/// Read integer values on RC
FUNCTION_BLOCK ReadIntegersFB EXTENDS RobotLibraryBaseFB
// ------------------------------------------------------------------------- 
//  SRCI Robot Library                                                
// ------------------------------------------------------------------------- 
//                                                                           
//  Object:      ReadIntegersFB                                       
//  Author:      Thorsten Brach                                                
//  Date:        2024-06-01
//
//  Description:                                              
//   
//                                                                           
//  Copyright: 
//    (C) 2024 Thorsten Brach. All rights reserved                                                                         
//                                                                           
//  Disclaimer:                                                                           
//    This project is provided without any guarantee and can be used for   
//    private and commercial purposes. Any commercial use is at the user’s 
//    own risk and responsibility.
//
// -------------------------------------------------------------------------
VAR_INPUT
  /// Start of the command at the rising edge
  Execute            : BOOL;
  /// Processing Mode
  ProcessingMode     : ProcessingMode;
  /// Specifies the desired target values that shall be read
  Index              : ARRAY[0..6] OF USINT; 
  /// Defines the target sequence in which the command will be executed
  SequenceFlag       : SequenceFlag;
  /// ID of associated trigger function:
  /// •  0: No Trigger (default)  No trigger related behavior
  /// • >0: Trigger - Start executing when the trigger function with the identical EmitterID is triggered.
  /// Always positive.
  /// For more information, see chapter 5.5.12 Triggers
  ListenerID         : SINT;
END_VAR
VAR_OUTPUT
  /// The command has been completed successfully
  Done               : BOOL;
  /// TRUE, while the following outputs return valid values:
  /// • Values
  Valid              : BOOL; 
  /// FB is being processed
  Busy               : BOOL;
  /// Command is transferred and confirmed by the RC
  CommandBuffered    : BOOL;
  /// The command was aborted by another command.
  CommandAborted     : BOOL;
  /// TRUE, while command is interrupted during execution and can be continued
  CommandInterrupted : BOOL;
  /// Receiving of input parameter values has been acknowledged by RC
  ParameterAccepted  : BOOL;
  /// Returned values of integer register
  Values             : ARRAY[0..6] OF INT;
  /// Unique system-generated ID of the "Action" when the function is triggered.
  /// • >0: The "Action" is started by the trigger function with identical FollowID.
  /// • <0: The "Action" is stopped by the trigger function with identical FollowID.
  /// For more information see chapter 5.5.12.4.
  OriginID           : USINT;
  /// Relates to ListenerID >0 
  /// Number of successful trigger -based command invocations
  /// For more information refer to chapter 5.5.12.4.
  InvocationCounter  : USINT;
END_VAR

                  
                

METHOD PROTECTED OnCall
VAR_IN_OUT
  /// Robot assignment of function
  AxesGroup         : AxesGroup; 
END_VAR
                        
                      
END_METHOD
END_FUNCTION_BLOCK

/// Read content of selected payload number
FUNCTION_BLOCK ReadLoadDataFB EXTENDS RobotLibraryBaseFB
// ------------------------------------------------------------------------- 
//  SRCI Robot Library                                                
// ------------------------------------------------------------------------- 
//                                                                           
//  Object:      ReadLoadDataFB                                       
//  Author:      Thorsten Brach                                                
//  Date:        2024-06-01
//
//  Description:                                              
//   
//                                                                           
//  Copyright: 
//    (C) 2024 Thorsten Brach. All rights reserved                                                                         
//                                                                           
//  Disclaimer:                                                                           
//    This project is provided without any guarantee and can be used for   
//    private and commercial purposes. Any commercial use is at the user’s 
//    own risk and responsibility.
//
// -------------------------------------------------------------------------
VAR_INPUT
  /// Start of the command at the rising edge
  Execute            : BOOL;
  /// Load index
  /// • -1: Currently used load on RC
  /// •  0: Not possible to read
  /// •  1 (default)..254: Load data
  LoadNo             : INT;
END_VAR
VAR_OUTPUT
  /// The command has been completed successfully
  Done               : BOOL;
  /// FB is being processed
  Busy               : BOOL;
  /// Command is transferred and confirmed by the RC
  CommandBuffered    : BOOL;
  /// Tool index
  LoadNoReturn       : USINT;
  /// Load data (see chapter 5.5.6.4)
  LoadData           : LoadData;
END_VAR

                  
                

METHOD PROTECTED OnCall
VAR_IN_OUT
  /// Robot assignment of function
  AxesGroup         : AxesGroup; 
END_VAR
                        
                      
END_METHOD
END_FUNCTION_BLOCK

/// Read error codes of pending errors and move them into user data block "RobotData"
FUNCTION_BLOCK ReadMessagesFB EXTENDS RobotLibraryBaseFB
// ------------------------------------------------------------------------- 
//  SRCI Robot Library                                                
// ------------------------------------------------------------------------- 
//                                                                           
//  Object:      ReadMessagesFB                                       
//  Author:      Thorsten Brach                                                
//  Date:        2024-06-01
//
//  Description:                                              
//   
//                                                                           
//  Copyright: 
//    (C) 2024 Thorsten Brach. All rights reserved                                                                         
//                                                                           
//  Disclaimer:                                                                           
//    This project is provided without any guarantee and can be used for   
//    private and commercial purposes. Any commercial use is at the user’s 
//    own risk and responsibility.
//
// -------------------------------------------------------------------------
VAR_INPUT
END_VAR
VAR_OUTPUT
END_VAR

                  
                

METHOD PROTECTED OnCall
VAR_IN_OUT
  /// Robot assignment of function
  AxesGroup         : AxesGroup; 
END_VAR
                        
                      
END_METHOD
END_FUNCTION_BLOCK

/// Read real values on RC
FUNCTION_BLOCK ReadRealsFB EXTENDS RobotLibraryBaseFB
// ------------------------------------------------------------------------- 
//  SRCI Robot Library                                                
// ------------------------------------------------------------------------- 
//                                                                           
//  Object:      ReadRealsFB                                       
//  Author:      Thorsten Brach                                                
//  Date:        2024-06-01
//
//  Description:                                              
//   
//                                                                           
//  Copyright: 
//    (C) 2024 Thorsten Brach. All rights reserved                                                                         
//                                                                           
//  Disclaimer:                                                                           
//    This project is provided without any guarantee and can be used for   
//    private and commercial purposes. Any commercial use is at the user’s 
//    own risk and responsibility.
//
// -------------------------------------------------------------------------
VAR_INPUT
  /// Start of the command at the rising edge
  Execute            : BOOL;
  /// Processing Mode
  ProcessingMode     : ProcessingMode;
  /// Specifies the desired target values that shall be read
  Index              : ARRAY[0..6] OF USINT; 
  /// Defines the target sequence in which the command will be executed
  SequenceFlag       : SequenceFlag;
  /// ID of associated trigger function:
  /// •  0: No Trigger (default)  No trigger related behavior
  /// • >0: Trigger - Start executing when the trigger function with the identical EmitterID is triggered.
  /// Always positive.
  /// For more information, see chapter 5.5.12 Triggers
  ListenerID         : SINT;
END_VAR
VAR_OUTPUT
  /// The command has been completed successfully
  Done               : BOOL;
  /// TRUE, while the following outputs return valid values:
  /// • Values
  Valid              : BOOL; 
  /// FB is being processed
  Busy               : BOOL;
  /// Command is transferred and confirmed by the RC
  CommandBuffered    : BOOL;
  /// The command was aborted by another command.
  CommandAborted     : BOOL;
  /// TRUE, while command is interrupted during execution and can be continued
  CommandInterrupted : BOOL;
  /// Receiving of input parameter values has been acknowledged by RC
  ParameterAccepted  : BOOL;
  /// Returned values of real register
  Values             : ARRAY[0..6] OF REAL;
  /// Unique system-generated ID of the "Action" when the function is triggered.
  /// • >0: The "Action" is started by the trigger function with identical FollowID.
  /// • <0: The "Action" is stopped by the trigger function with identical FollowID.
  /// For more information see chapter 5.5.12.4.
  OriginID           : USINT;
  /// Relates to ListenerID >0 
  /// Number of successful trigger -based command invocations
  /// For more information refer to chapter 5.5.12.4.
  InvocationCounter  : USINT;
END_VAR

                  
                

METHOD PROTECTED OnCall
VAR_IN_OUT
  /// Robot assignment of function
  AxesGroup         : AxesGroup; 
END_VAR
                        
                      
END_METHOD
END_FUNCTION_BLOCK

/// Read robot-specific data from the RC
FUNCTION_BLOCK ReadRobotDataFB EXTENDS RobotLibraryBaseFB
// ------------------------------------------------------------------------- 
//  SRCI Robot Library                                                
// ------------------------------------------------------------------------- 
//                                                                           
//  Object:      ReadRobotDataFB                                       
//  Author:      Thorsten Brach                                                
//  Date:        2024-06-01
//
//  Description:                                              
//   
//                                                                           
//  Copyright: 
//    (C) 2024 Thorsten Brach. All rights reserved                                                                         
//                                                                           
//  Disclaimer:                                                                           
//    This project is provided without any guarantee and can be used for   
//    private and commercial purposes. Any commercial use is at the user’s 
//    own risk and responsibility.
//
// -------------------------------------------------------------------------
VAR_INPUT
END_VAR
VAR_OUTPUT
END_VAR

                  
                

METHOD PROTECTED OnCall
VAR_IN_OUT
  /// Robot assignment of function
  AxesGroup         : AxesGroup; 
END_VAR
                        
                      
END_METHOD
END_FUNCTION_BLOCK

/// Read default values of dynamic parameters used by move commands
FUNCTION_BLOCK ReadRobotDefaultDynamicsFB EXTENDS RobotLibraryBaseFB
// ------------------------------------------------------------------------- 
//  SRCI Robot Library                                                
// ------------------------------------------------------------------------- 
//                                                                           
//  Object:      ReadRobotDefaultDynamicsFB                                       
//  Author:      Thorsten Brach                                                
//  Date:        2024-06-01
//
//  Description:                                              
//   
//                                                                           
//  Copyright: 
//    (C) 2024 Thorsten Brach. All rights reserved                                                                         
//                                                                           
//  Disclaimer:                                                                           
//    This project is provided without any guarantee and can be used for   
//    private and commercial purposes. Any commercial use is at the user’s 
//    own risk and responsibility.
//
// -------------------------------------------------------------------------
VAR_INPUT
  /// Start of the command at the rising edge
  Execute            : BOOL;
END_VAR

VAR_OUTPUT
  /// The command has been completed successfully
  Done               : BOOL;
  /// FB is being processed
  Busy               : BOOL;
  /// Command is transferred and confirmed by the RC
  CommandBuffered    : BOOL;
  /// Default dynamics values according to Table 6-148.
  DynamicValues      : DefaultDynamics;
END_VAR

                  
                

METHOD PROTECTED OnCall
VAR_IN_OUT
  /// Robot assignment of function
  AxesGroup         : AxesGroup; 
END_VAR
                        
                      
END_METHOD
END_FUNCTION_BLOCK

/// Read reference values of robot dynamics for path movement
FUNCTION_BLOCK ReadRobotReferenceDynamicsFB EXTENDS RobotLibraryBaseFB
// ------------------------------------------------------------------------- 
//  SRCI Robot Library                                                
// ------------------------------------------------------------------------- 
//                                                                           
//  Object:      ReadRobotReferenceDynamicsFB                                       
//  Author:      Thorsten Brach                                                
//  Date:        2024-06-01
//
//  Description:                                              
//   
//                                                                           
//  Copyright: 
//    (C) 2024 Thorsten Brach. All rights reserved                                                                         
//                                                                           
//  Disclaimer:                                                                           
//    This project is provided without any guarantee and can be used for   
//    private and commercial purposes. Any commercial use is at the user’s 
//    own risk and responsibility.
//
// -------------------------------------------------------------------------
VAR_INPUT
  /// Start of the command at the rising edge
  Execute            : BOOL;
END_VAR

VAR_OUTPUT
  /// The command has been completed successfully
  Done               : BOOL;
  /// FB is being processed
  Busy               : BOOL;
  /// Command is transferred and confirmed by the RC
  CommandBuffered    : BOOL;
  /// Reference dynamics values according to Table 6-109.
  DynamicValues      : ReferenceDynamics;
END_VAR

                  
                

METHOD PROTECTED OnCall
VAR_IN_OUT
  /// Robot assignment of function
  AxesGroup         : AxesGroup; 
END_VAR
                        
                      
END_METHOD
END_FUNCTION_BLOCK

/// Read actual software limits of the axes Positive and negative Limit of Joint J1…J6, E1…E6
FUNCTION_BLOCK ReadRobotSWLimitsFB EXTENDS RobotLibraryBaseFB
// ------------------------------------------------------------------------- 
//  SRCI Robot Library                                                
// ------------------------------------------------------------------------- 
//                                                                           
//  Object:      ReadRobotSWLimitsFB                                       
//  Author:      Thorsten Brach                                                
//  Date:        2024-06-01
//
//  Description:                                              
//   
//                                                                           
//  Copyright: 
//    (C) 2024 Thorsten Brach. All rights reserved                                                                         
//                                                                           
//  Disclaimer:                                                                           
//    This project is provided without any guarantee and can be used for   
//    private and commercial purposes. Any commercial use is at the user’s 
//    own risk and responsibility.
//
// -------------------------------------------------------------------------
VAR_INPUT
  /// Start of the command at the rising edge
  Execute            : BOOL;
END_VAR

VAR_OUTPUT
  /// The command has been completed successfully
  Done               : BOOL;
  /// FB is being processed
  Busy               : BOOL;
  /// Command is transferred and confirmed by the RC
  CommandBuffered    : BOOL;
  /// DLimits for joints and external axes according to Table 6-173.
  LimitValues        : SWLimits;
END_VAR

                  
                

METHOD PROTECTED OnCall
VAR_IN_OUT
  /// Robot assignment of function
  AxesGroup         : AxesGroup; 
END_VAR
                        
                      
END_METHOD
END_FUNCTION_BLOCK

/// Read specific parameter of the robot
FUNCTION_BLOCK ReadSystemVariableFB EXTENDS RobotLibraryBaseFB
// ------------------------------------------------------------------------- 
//  SRCI Robot Library                                                
// ------------------------------------------------------------------------- 
//                                                                           
//  Object:      ReadSystemVariableFB                                       
//  Author:      Thorsten Brach                                                
//  Date:        2024-06-01
//
//  Description:                                              
//   
//                                                                           
//  Copyright: 
//    (C) 2024 Thorsten Brach. All rights reserved                                                                         
//                                                                           
//  Disclaimer:                                                                           
//    This project is provided without any guarantee and can be used for   
//    private and commercial purposes. Any commercial use is at the user’s 
//    own risk and responsibility.
//
// -------------------------------------------------------------------------
VAR_INPUT
  /// Start of the command at the rising edge
  Execute            : BOOL;
  /// Processing Mode
  ProcessingMode     : ProcessingMode;
  /// Defines the parameter list which should be used:
  /// • FALSE: Standardized parameter list (default):
  ///          -  Read parameters on the RC based on a standardized parameter list
  /// • TRUE: Manufacturer specific parameter list:
  ///        -  Read parameters on the RC based on robot manufacturers-specific parameter lists
  RCParameter        : BOOL;
  /// Requested parameter ID in selected parameter list.
  /// •          0: undefined (default)
  /// • 1..65 535: Parameter ID
  ParameterID        : ARRAY[0..7] OF UINT;
  /// ID of the requested sub parameter in selected parameter list.
  /// • 0: ID 0 (default) (relates only to parameters without sub parameters)
  /// • 1..255: Indices 1 to 255 (relates only to parameters with sub parameters)
  SubParameterID     : ARRAY[0..7] OF USINT;
  /// Defines the target sequence in which the command will be executed
  SequenceFlag       : SequenceFlag;
  /// ID of associated trigger function:
  /// •  0: No Trigger (default)  No trigger related behavior
  /// • >0: Trigger - Start executing when the trigger function with the identical EmitterID is triggered.
  /// Always positive.
  /// For more information, see chapter 5.5.12 Triggers
  ListenerID         : SINT;
END_VAR
VAR_OUTPUT
  /// The command has been completed successfully
  Done               : BOOL;
  /// TRUE, while the following outputs return valid values:
  /// • DataType
  /// • Data_0
  /// • Data_1
  /// • Data_2
  /// • Data_3
  /// • Data_4
  /// • Data_5
  /// • Data_6
  /// • Data_7
  Valid              : BOOL; 
  /// FB is being processed
  Busy               : BOOL;
  /// Command is transferred and confirmed by the RC
  CommandBuffered    : BOOL;
  /// The command was aborted by another command.
  CommandAborted     : BOOL;
  /// TRUE, while command is interrupted during execution and can be continued
  CommandInterrupted : BOOL;
  /// Receiving of input parameter values has been acknowledged by RC
  ParameterAccepted  : BOOL;
  /// Parameter data type as specified in Table 6-613.
  DataType           : ARRAY[0..7] OF USINT;
  /// Parameter data addressed by input values of ParameterID[0] and SubParameterID[0]
  Data_0             : ARRAY[0..3] OF BYTE;
  /// Parameter data addressed by input values of ParameterID[1] and SubParameterID[1]
  Data_1             : ARRAY[0..3] OF BYTE;
  /// Parameter data addressed by input values of ParameterID[2] and SubParameterID[2]
  Data_2             : ARRAY[0..3] OF BYTE;
  /// Parameter data addressed by input values of ParameterID[3] and SubParameterID[3]
  Data_3             : ARRAY[0..3] OF BYTE;
  /// Parameter data addressed by input values of ParameterID[4] and SubParameterID[4]
  Data_4             : ARRAY[0..3] OF BYTE;
  /// Parameter data addressed by input values of ParameterID[5] and SubParameterID[5]
  Data_5             : ARRAY[0..3] OF BYTE;
  /// Parameter data addressed by input values of ParameterID[6] and SubParameterID[6]
  Data_6             : ARRAY[0..3] OF BYTE;
  /// Parameter data addressed by input values of ParameterID[7] and SubParameterID[7]
  Data_7             : ARRAY[0..3] OF BYTE;
  /// Unique system-generated ID of the "Action" when the function is triggered.
  /// • >0: The "Action" is started by the trigger function with identical FollowID.
  /// • <0: The "Action" is stopped by the trigger function with identical FollowID.
  /// For more information see chapter 5.5.12.4 EmitterID, ListenerID, FollowID and OriginID
  OriginID           : INT;
  /// Relates to ListenerID >0
  /// Number of successful trigger -based command invocations
  /// For more information refer to chapter 5.5.12.4.
  InvocationCounter  : USINT;
END_VAR

                  
                

METHOD PROTECTED OnCall
VAR_IN_OUT
  /// Robot assignment of function
  AxesGroup         : AxesGroup; 
END_VAR
                        
                      
END_METHOD
END_FUNCTION_BLOCK

/// Read content of selected tool number
FUNCTION_BLOCK ReadToolDataFB EXTENDS RobotLibraryBaseFB
// ------------------------------------------------------------------------- 
//  SRCI Robot Library                                                
// ------------------------------------------------------------------------- 
//                                                                           
//  Object:      ReadToolDataFB                                       
//  Author:      Thorsten Brach                                                
//  Date:        2024-06-01
//
//  Description:                                              
//   
//                                                                           
//  Copyright: 
//    (C) 2024 Thorsten Brach. All rights reserved                                                                         
//                                                                           
//  Disclaimer:                                                                           
//    This project is provided without any guarantee and can be used for   
//    private and commercial purposes. Any commercial use is at the user’s 
//    own risk and responsibility.
//
// -------------------------------------------------------------------------
VAR_INPUT
  /// Start of the command at the rising edge
  Execute            : BOOL;
  /// Tool index
  /// • -1: Currently used tool on RC
  /// •  0: Flange -  Not possible to change
  /// • 1 (default)..254: Tool Frame
  ToolNo             : INT;
END_VAR
VAR_OUTPUT
  /// The command has been completed successfully
  Done               : BOOL;
  /// FB is being processed
  Busy               : BOOL;
  /// Command is transferred and confirmed by the RC
  CommandBuffered    : BOOL;
  /// Tool index
  ToolNoReturn       : USINT;
  /// Tool data (see chapter 5.5.6.3)
  ToolData           : ToolData;
END_VAR

                  
                

METHOD PROTECTED OnCall
VAR_IN_OUT
  /// Robot assignment of function
  AxesGroup         : AxesGroup; 
END_VAR
                        
                      
END_METHOD
END_FUNCTION_BLOCK

/// Read configuration of defined work areas
FUNCTION_BLOCK ReadWorkAreaFB EXTENDS RobotLibraryBaseFB
// ------------------------------------------------------------------------- 
//  SRCI Robot Library                                                
// ------------------------------------------------------------------------- 
//                                                                           
//  Object:      ReadWorkAreaFB                                       
//  Author:      Thorsten Brach                                                
//  Date:        2024-06-01
//
//  Description:                                              
//   
//                                                                           
//  Copyright: 
//    (C) 2024 Thorsten Brach. All rights reserved                                                                         
//                                                                           
//  Disclaimer:                                                                           
//    This project is provided without any guarantee and can be used for   
//    private and commercial purposes. Any commercial use is at the user’s 
//    own risk and responsibility.
//
// -------------------------------------------------------------------------
VAR_INPUT
  /// Start of the command at the rising edge
  Execute                : BOOL;
  /// Index of the robot work area
  /// • 0 (default)..254
  WorkAreaNo             : USINT;
END_VAR
VAR_OUTPUT
  /// The command has been completed successfully
  Done                   : BOOL;
  /// FB is being processed
  Busy                   : BOOL;
  /// Command is transferred and confirmed by the RC
  CommandBuffered        : BOOL;
  /// Index of the robot work area
  WorkAreaNoReturn       : USINT;
  /// Data specific to the work area requested by Index.
  WorkAreaData           : RobotWorkArea;
END_VAR

                  
                

METHOD PROTECTED OnCall
VAR_IN_OUT
  /// Robot assignment of function
  AxesGroup         : AxesGroup; 
END_VAR
                        
                      
END_METHOD
END_FUNCTION_BLOCK

/// Move robot into contact with obstruction (mechanical Limit) and hold it in this position
FUNCTION_BLOCK SearchHardStopFB EXTENDS RobotLibraryBaseFB
// ------------------------------------------------------------------------- 
//  SRCI Robot Library                                                
// ------------------------------------------------------------------------- 
//                                                                           
//  Object:      SearchHardStopFB                                       
//  Author:      Thorsten Brach                                                
//  Date:        2024-06-01
//
//  Description:                                              
//   
//                                                                           
//  Copyright: 
//    (C) 2024 Thorsten Brach. All rights reserved                                                                         
//                                                                           
//  Disclaimer:                                                                           
//    This project is provided without any guarantee and can be used for   
//    private and commercial purposes. Any commercial use is at the user’s 
//    own risk and responsibility.
//
// -------------------------------------------------------------------------
VAR_INPUT
  /// Start of the command at the rising edge
  Execute            : BOOL;
  /// Absolute target coordinates in the selected coordinate system (see input parameters ToolNo and FrameNo)
  Position           : RobotCartesianPosition;
  /// Defines the type of collision detection, which parameter should be observed
  DetectionMode      : DetectionMode;
  /// Additional parameter for the detection of an end position. Defines the limits for seven joints, 
  /// where the robot stops when one of the limits is reached. Unit is depending on the "DetectionMode":
  /// • Torque (default) [Nm]  - Only positive values accepted
  /// • Force [N]              - Only positive values accepted
  /// • Electrical current [A] - Only positive values accepted
  /// • Following Error [mm]   - >0: Robot stops when the following error reached positive limit
  ///                          - <0: Robot stops when the following error reaches the negative limit
  DetectionVector    : ARRAY [0..6] OF REAL;
  /// TCP velocity in % of nominal velocity
  /// •  <0%: (default) - Use default velocity
  /// •   0%:           - Use internal minimal velocity
  /// • 100%:           - Use maximal reference velocity
  /// See chapter 5.5.7 Robot dynamics
  VelocityRate       : REAL;
  /// Acceleration for movement in % of nominal acceleration
  /// •  <0%: (default) - Use default acceleration
  /// •   0%:           - Use internal minimal acceleration
  /// • 100%:           - Use maximal reference acceleration
  /// See chapter 5.5.7 Robot dynamics
  AccelerationRate   : REAL;
  /// Deceleration for movement in % of nominal deceleration
  /// •  <0%: (default) - Use default deceleration 
  /// •   0%:           - Use internal minimal deceleration
  /// • 100%:           - Use maximal reference deceleration
  /// See chapter 5.5.7 Robot dynamics
  DecelerationRate   : REAL;
  /// Jerk of the movement in % of nominal jerk
  /// •  <0%: (default) - Use default jerk
  /// •   0%:           - Use internal minimal jerk
  /// • 100%:           - Use maximal reference jerk
  /// See chapter 5.5.7 Robot dynamics
  JerkRate           : REAL;
  /// Index of tool
  /// •      0: Flange (default)
  /// • 1..254: Tool frames
  ToolNo             : USINT;
  /// Index of frame
  /// •      0: WCS (default)
  /// • 1..254: User frames
  FrameNo            : USINT;
  /// Parameter which determines the behavior towards the previously sent and still active or buffered commands
  AbortingMode       : AbortingMode;
  /// Parameter to describe how the orientation axes (RX, RY, RZ) will be interpolated during the movement
  OriMode            : OriMode;
  /// Defines the usage of the config byte inside the position according to Table 6-238
  ConfigMode         : ArmConfigParameter;
  /// Defines the usage of the TurnNumber byte inside the position.
  TurnMode           : TurnMode;
  /// Set TRUE to allow manipulation of this move command through superimposing functions.
  /// For more information see chapter 5.5.9.5
  Manipulation       : BOOL;
  /// Defines the target sequence in which the command will be executed
  SequenceFlag       : SequenceFlag;
END_VAR

VAR_OUTPUT
  /// The command has been completed successfully
  Done               : BOOL;
  /// FB is being processed
  Busy               : BOOL;
  /// Command is transferred and confirmed by the RC
  CommandBuffered    : BOOL;
  /// The command takes control of the motion of the according axis group
  Active             : BOOL;
  /// The command was aborted by another command.
  CommandAborted     : BOOL;
  /// TRUE, while command is interrupted during execution and can be continued
  CommandInterrupted : BOOL;
  /// Distance-to-go of the current job.
  /// • -1: No valid value because move command is not yet active (valid values are pending) or not supported by RC
  /// • >0: Actual distance between current and target position
  /// •  0: Target position reached
  RemainingDistance  : REAL;
  /// Percentage of already traversed distance of current job.
  /// If not supported : • -1
  Progress           : REAL;
  /// The robot arm has detected an obstruction and stopped the movement
  InClamping         : BOOL;
END_VAR

                  
                

METHOD PROTECTED OnCall
VAR_IN_OUT
  /// Robot assignment of function
  AxesGroup         : AxesGroup; 
END_VAR
                        
                      
END_METHOD
END_FUNCTION_BLOCK

/// Move robot into contact with obstruction (mechanical Limit) and hold it in this position
FUNCTION_BLOCK SearchHardStopJFB EXTENDS RobotLibraryBaseFB
// ------------------------------------------------------------------------- 
//  SRCI Robot Library                                                
// ------------------------------------------------------------------------- 
//                                                                           
//  Object:      SearchHardStopJFB                                       
//  Author:      Thorsten Brach                                                
//  Date:        2024-06-01
//
//  Description:                                              
//   
//                                                                           
//  Copyright: 
//    (C) 2024 Thorsten Brach. All rights reserved                                                                         
//                                                                           
//  Disclaimer:                                                                           
//    This project is provided without any guarantee and can be used for   
//    private and commercial purposes. Any commercial use is at the user’s 
//    own risk and responsibility.
//
// -------------------------------------------------------------------------
VAR_INPUT
  /// Start of the command at the rising edge
  Execute            : BOOL;
  /// Absolute target coordinates in the selected coordinate system (see input parameters ToolNo and FrameNo)
  JointPosition      : RobotJointPosition;
  /// Defines the type of collision detection, which parameter should be observed
  DetectionMode      : DetectionMode;
  /// Additional parameter for the detection of an end position. Defines the limits for seven joints, 
  /// where the robot stops when one of the limits is reached. Unit is depending on the "DetectionMode":
  /// • Torque (default) [Nm]  - Only positive values accepted
  /// • Force [N]              - Only positive values accepted
  /// • Electrical current [A] - Only positive values accepted
  /// • Following Error [mm]   - >0: Robot stops when the following error reached positive limit
  ///                          - <0: Robot stops when the following error reaches the negative limit
  DetectionVector    : ARRAY [0..6] OF REAL;
  /// TCP velocity in % of nominal velocity
  /// •  <0%: (default) - Use default velocity
  /// •   0%:           - Use internal minimal velocity
  /// • 100%:           - Use maximal reference velocity
  /// See chapter 5.5.7 Robot dynamics
  VelocityRate       : REAL;
  /// Acceleration for movement in % of nominal acceleration
  /// •  <0%: (default) - Use default acceleration
  /// •   0%:           - Use internal minimal acceleration
  /// • 100%:           - Use maximal reference acceleration
  /// See chapter 5.5.7 Robot dynamics
  AccelerationRate   : REAL;
  /// Deceleration for movement in % of nominal deceleration
  /// •  <0%: (default) - Use default deceleration 
  /// •   0%:           - Use internal minimal deceleration
  /// • 100%:           - Use maximal reference deceleration
  /// See chapter 5.5.7 Robot dynamics
  DecelerationRate   : REAL;
  /// Jerk of the movement in % of nominal jerk
  /// •  <0%: (default) - Use default jerk
  /// •   0%:           - Use internal minimal jerk
  /// • 100%:           - Use maximal reference jerk
  /// See chapter 5.5.7 Robot dynamics
  JerkRate           : REAL;
  /// Index of tool
  /// •      0: Flange (default)
  /// • 1..254: Tool frames
  ToolNo             : USINT;
  /// Parameter which determines the behavior towards the previously sent and still active or buffered commands
  AbortingMode       : AbortingMode;
  /// Set TRUE to allow manipulation of this move command through superimposing functions.
  /// For more information see chapter 5.5.9.5
  Manipulation       : BOOL;
  /// Defines the target sequence in which the command will be executed
  SequenceFlag       : SequenceFlag;
END_VAR

VAR_OUTPUT
  /// The command has been completed successfully
  Done               : BOOL;
  /// FB is being processed
  Busy               : BOOL;
  /// Command is transferred and confirmed by the RC
  CommandBuffered    : BOOL;
  /// The command takes control of the motion of the according axis group
  Active             : BOOL;
  /// The command was aborted by another command.
  CommandAborted     : BOOL;
  /// TRUE, while command is interrupted during execution and can be continued
  CommandInterrupted : BOOL;
  /// Distance-to-go of the current job.
  /// • -1: No valid value because move command is not yet active (valid values are pending) or not supported by RC
  /// • >0: Actual distance between current and target position
  /// •  0: Target position reached
  RemainingDistance  : REAL;
  /// Percentage of already traversed distance of current job.
  /// If not supported : • -1
  Progress           : REAL;
  /// The robot arm has detected an obstruction and stopped the movement
  InClamping         : BOOL;
END_VAR

                  
                

METHOD PROTECTED OnCall
VAR_IN_OUT
  /// Robot assignment of function
  AxesGroup         : AxesGroup; 
END_VAR
                        
                      
END_METHOD
END_FUNCTION_BLOCK

/// Switch operation mode of RC (Automatic External, T1 External, T2 External)
FUNCTION_BLOCK SetOperationModeFB EXTENDS RobotLibraryBaseFB
// ------------------------------------------------------------------------- 
//  SRCI Robot Library                                                
// ------------------------------------------------------------------------- 
//                                                                           
//  Object:      SetOperationModeFB                                       
//  Author:      Thorsten Brach                                                
//  Date:        2024-06-01
//
//  Description:                                              
//   
//                                                                           
//  Copyright: 
//    (C) 2024 Thorsten Brach. All rights reserved                                                                         
//                                                                           
//  Disclaimer:                                                                           
//    This project is provided without any guarantee and can be used for   
//    private and commercial purposes. Any commercial use is at the user’s 
//    own risk and responsibility.
//
// -------------------------------------------------------------------------
VAR_INPUT
  /// Start of the command at the rising edge
  Execute                : BOOL;
  /// Limits for joints and external axes according to Table 6-180.
  OperationMode           : OperationMode;
END_VAR
VAR_OUTPUT
  /// The command has been completed successfully
  Done                   : BOOL;
  /// FB is being processed
  Busy                   : BOOL;
  /// Command is transferred and confirmed by the RC
  CommandBuffered        : BOOL;
END_VAR

                  
                

METHOD PROTECTED OnCall
VAR_IN_OUT
  /// Robot assignment of function
  AxesGroup         : AxesGroup; 
END_VAR
                        
                      
END_METHOD
END_FUNCTION_BLOCK

/// Set active sequence
FUNCTION_BLOCK SetSequenceFB EXTENDS RobotLibraryBaseFB
// ------------------------------------------------------------------------- 
//  SRCI Robot Library                                                
// ------------------------------------------------------------------------- 
//                                                                           
//  Object:      SetSequenceFB                                       
//  Author:      Thorsten Brach                                                
//  Date:        2024-06-01
//
//  Description:                                              
//   
//                                                                           
//  Copyright: 
//    (C) 2024 Thorsten Brach. All rights reserved                                                                         
//                                                                           
//  Disclaimer:                                                                           
//    This project is provided without any guarantee and can be used for   
//    private and commercial purposes. Any commercial use is at the user’s 
//    own risk and responsibility.
//
// -------------------------------------------------------------------------
VAR_INPUT
  /// Start of the command at the rising edge
  Execute         : BOOL;
  /// Defines sequence to be activated when function is executed
  TargetSequence  : SequenceFlag;
END_VAR

VAR_OUTPUT
  /// The command has been completed successfully
  Done            : BOOL;
  /// FB is being processed
  Busy            : BOOL;
  /// Command is transferred and confirmed by the RC
  CommandBuffered : BOOL;
END_VAR

                  
                

METHOD PROTECTED OnCall
VAR_IN_OUT
  /// Robot assignment of function
  AxesGroup         : AxesGroup; 
END_VAR
                        
                      
END_METHOD
END_FUNCTION_BLOCK

/// Create spline on RC from positions stored in PLC
FUNCTION_BLOCK CreateSplineFB EXTENDS RobotLibraryBaseFB
// ------------------------------------------------------------------------- 
//  SRCI Robot Library                                                
// ------------------------------------------------------------------------- 
//                                                                           
//  Object:      CreateSplineFB                                       
//  Author:      Thorsten Brach                                                
//  Date:        2024-06-01
//
//  Description:                                              
//   
//                                                                           
//  Copyright: 
//    (C) 2024 Thorsten Brach. All rights reserved                                                                         
//                                                                           
//  Disclaimer:                                                                           
//    This project is provided without any guarantee and can be used for   
//    private and commercial purposes. Any commercial use is at the user’s 
//    own risk and responsibility.
//
// -------------------------------------------------------------------------
VAR_INPUT
  /// Start of the command at the rising edge
  Execute         : BOOL;
  /// Define the method to calculate the path trajectory for the spline movement
  Mode            : SplineMode;
  /// Index of the spline trajectory to be created
  SplineID        : SINT;
  /// Contains all data relevant to the spline trajectory
  /// • Cartesian position
  /// • Coordinate systems
  /// • Dynamic parameters
  /// For more information refer to chapter 5.5.13.3
  SplineData      : ARRAY[1..RobotLibraryParameter.SPLINE_DATA_MAX] OF SplineData;
END_VAR
VAR_OUTPUT
  /// The command has been completed successfully
  Done            : BOOL;
  /// FB is being processed
  Busy            : BOOL;
  /// Command is transferred and confirmed by the RC
  CommandBuffered : BOOL;
END_VAR

                  
                

METHOD PROTECTED OnCall
VAR_IN_OUT
  /// Robot assignment of function
  AxesGroup         : AxesGroup; 
END_VAR
                        
                      
END_METHOD
END_FUNCTION_BLOCK

/// Delete spline previously created on RC
FUNCTION_BLOCK DeleteSplineFB EXTENDS RobotLibraryBaseFB
// ------------------------------------------------------------------------- 
//  SRCI Robot Library                                                
// ------------------------------------------------------------------------- 
//                                                                           
//  Object:      DeleteSplineFB                                       
//  Author:      Thorsten Brach                                                
//  Date:        2024-06-01
//
//  Description:                                              
//   
//                                                                           
//  Copyright: 
//    (C) 2024 Thorsten Brach. All rights reserved                                                                         
//                                                                           
//  Disclaimer:                                                                           
//    This project is provided without any guarantee and can be used for   
//    private and commercial purposes. Any commercial use is at the user’s 
//    own risk and responsibility.
//
// -------------------------------------------------------------------------
VAR_INPUT
  /// Start of the command at the rising edge
  Execute         : BOOL;
  /// Index of the spline trajectory to be deleted
  SplineID        : SINT;
END_VAR
VAR_OUTPUT
  /// The command has been completed successfully
  Done            : BOOL;
  /// FB is being processed
  Busy            : BOOL;
  /// Command is transferred and confirmed by the RC
  CommandBuffered : BOOL;
END_VAR

                  
                

METHOD PROTECTED OnCall
VAR_IN_OUT
  /// Robot assignment of function
  AxesGroup         : AxesGroup; 
END_VAR
                        
                      
END_METHOD
END_FUNCTION_BLOCK

/// Create and move spline on RC simultaneously
FUNCTION_BLOCK DynamicSplineFB EXTENDS RobotLibraryBaseFB
// ------------------------------------------------------------------------- 
//  SRCI Robot Library                                                
// ------------------------------------------------------------------------- 
//                                                                           
//  Object:      DynamicSplineFB                                       
//  Author:      Thorsten Brach                                                
//  Date:        2024-06-01
//
//  Description:                                              
//   
//                                                                           
//  Copyright: 
//    (C) 2024 Thorsten Brach. All rights reserved                                                                         
//                                                                           
//  Disclaimer:                                                                           
//    This project is provided without any guarantee and can be used for   
//    private and commercial purposes. Any commercial use is at the user’s 
//    own risk and responsibility.
//
// -------------------------------------------------------------------------
VAR_INPUT
  /// Start of the command at the rising edge
  Execute            : BOOL;
  /// Define the method to calculate the path trajectory for the spline movement
  Mode               : SplineMode;
  /// Parameter which determines the behavior towards the previously sent and still active or buffered commands
  AbortingMode       : AbortingMode;
  /// Parameter which determines the transition behavior at the end of the movement to be sent to the next command. 
  /// The user can choose a transition type between exact stop and different blend possibilities.
  BlendingMode       : BlendingMode;
  /// Additional parameter for the blending mode, to define i.e. velocity limit (%) or blending radius
  /// • [0]: default 10
  /// • [1]: default 0
  BlendingParameter  : ARRAY [0..1] OF REAL;
  /// Parameter is used if it is greater than 0 (default):
  /// • Velocity input is ignored
  /// • Parameter defines the time for the movement to reach the target position 
  /// Error is sent by the RC, if the time cannot be kept.
  MoveTime           : UINT;
  /// Contains all data relevant to the spline trajectory
  /// • Cartesian position
  /// • Coordinate systems
  /// • Dynamic parameters
  /// For more information refer to chapter 5.5.13.3
  SplineData         : ARRAY[1..RobotLibraryParameter.SPLINE_DATA_MAX] OF SplineData;
  /// Starts calculation and spline motion when equal or greater to number of buffered spline positions
  StartPosition      : INT; 
  /// Defines the target sequence in which the command will be executed
  SequenceFlag       : SequenceFlag;
END_VAR
VAR_OUTPUT
  /// FB is being processed
  Busy               : BOOL;
  /// Command is transferred and confirmed by the RC
  CommandBuffered    : BOOL;
  /// Function is enabled and new input values will be transmitted.
  Enabled            : BOOL;
  /// The command takes control of the motion of the according axis group
  Active             : BOOL;
  /// The command was aborted by another command.
  CommandAborted     : BOOL;
  /// TRUE, while command is interrupted during execution and can be continued.
  CommandInterrupted : BOOL;
  /// Receiving of input parameter values has been acknowledged by RC
  ParameterAccepted  : BOOL;
  /// Distance-to-go of the current job.
  /// • -1: No valid value because move command is not yet active (valid values are pending) or not supported by RC
  /// • >0: Actual distance between current and target position
  /// •  0: Target position reached 
  RemainingDistance  : REAL;
  /// Percentage of already traversed distance of actual segment of spline trajectory.
  /// If not supported: -1
  SegmentProgress    : REAL;
  /// Number of buffered, consecutive segments of spline trajectory. 
  Buffered           : INT;
  /// Number of calculated, consecutive segments of spline trajectory. Already calculated segments can no longer be modified.
  Calculated         : INT;
  /// Index of the currently active segment of spline data set.
  ActualIndex        : SINT;  
  /// Spline movement has been finished successfully. New SplineData will start a new spline movement.
  TrajectoryCompleted: BOOL;
END_VAR

                  
                

METHOD PROTECTED OnCall
VAR_IN_OUT
  /// Robot assignment of function
  AxesGroup         : AxesGroup; 
END_VAR
                        
                      
END_METHOD
END_FUNCTION_BLOCK

/// Call subprogram stored in RC from PLC
FUNCTION_BLOCK CallSubprogramFB EXTENDS RobotLibraryBaseFB
// ------------------------------------------------------------------------- 
//  SRCI Robot Library                                                
// ------------------------------------------------------------------------- 
//                                                                           
//  Object:      CallSubprogramFB                                       
//  Author:      Thorsten Brach                                                
//  Date:        2024-06-01
//
//  Description:                                              
//   
//                                                                           
//  Copyright: 
//    (C) 2024 Thorsten Brach. All rights reserved                                                                         
//                                                                           
//  Disclaimer:                                                                           
//    This project is provided without any guarantee and can be used for   
//    private and commercial purposes. Any commercial use is at the user’s 
//    own risk and responsibility.
//
// -------------------------------------------------------------------------
VAR_INPUT
  /// Start of the command at the rising edge
  Execute           : BOOL;
  /// Processing mode
  ProcessingMode    : ProcessingMode;
  /// Program number of the subprogram in the RC
  JobID             : UINT;
  /// Defines the target sequence in which the command will be executed
  SequenceFlag      : SequenceFlag;
  /// ID of associated trigger function:
  /// • 0: No Trigger (default) - No trigger related behavior
  /// • >0: Triggero - Start executing when the trigger function with the identical EmitterID is triggered.
  /// Always positive.
  /// For more information, see chapter 5.5.12 Triggers
  ListenerID        : SINT;
  /// Acyclic input parameters of the subprogram Array length adjusts to transmitted data (max 190 bytes)
  Data              : ARRAY[0..RobotLibraryParameter.SUB_PROGRAM_DATA_MAX] OF BYTE;
END_VAR

VAR_OUTPUT
  /// The command has been completed successfully
  Done               : BOOL;
  /// TRUE while the output ReturnData returns valid data according to the user defined subprogram
  Valid              : BOOL;
  /// FB is being processed
  Busy               : BOOL;
  /// Command is transferred and confirmed by the RC
  CommandBuffered    : BOOL;
  /// The requested subprogram on the RC is in progress. Movement of the axes trough this subprogram is possible.  
  InProgress         : BOOL;
  /// The command was aborted by another command
  CommandAborted     : BOOL;
  /// TRUE, while command is interrupted during execution and can be continued.
  CommandInterrupted : BOOL;
  /// Receiving of input parameter values has been acknowledged by RC
  ParameterAccepted  : BOOL;
  /// Unique, system-generated ID of the instance of CallSubprogram. 
  /// Can be used to specifically stop instance of a subprogram via the function Stop Subprogram (chapter 6.5.21) 
  /// if multiinstancing  is supported by RC 
  InstanceID         : DINT; 
  /// Percentage of already processed subprogram (must be configured by user)
  Progress           : REAL;
  /// Unique system-generated ID of the "Action" when the function is triggered.
  /// • >0: The "Action" is started by the trigger function with identical FollowID.
  /// • <0: The "Action" is stopped by the trigger function with identical FollowID.
  /// For more information see chapter 5.5.12.4 EmitterID, ListenerID, FollowID and OriginID
  OriginID           : INT;
  /// Relates to ListenerID >0
  /// Number of successful trigger -based command invocations
  /// For more information refer to chapter 5.5.12.4.
  InvocationCounter  : USINT;
  /// Acyclic output parameters of the subprogram Array length adjusts to transmitted data (max 190 bytes)
  ReturnData         : ARRAY[0..RobotLibraryParameter.SUB_PROGRAM_DATA_MAX] OF BYTE;
END_VAR

                  
                

METHOD PROTECTED OnCall
VAR_IN_OUT
  /// Robot assignment of function
  AxesGroup         : AxesGroup; 
END_VAR
                        
                      
END_METHOD
END_FUNCTION_BLOCK

/// Reads cyclic data of called subprogram
FUNCTION_BLOCK ReadCallSubprogramCyclicFB EXTENDS RobotLibraryBaseFB
// ------------------------------------------------------------------------- 
//  SRCI Robot Library                                                
// ------------------------------------------------------------------------- 
//                                                                           
//  Object:      ReadCallSubprogramCyclicFB                                       
//  Author:      Thorsten Brach                                                
//  Date:        2024-06-01
//
//  Description:                                              
//   
//                                                                           
//  Copyright: 
//    (C) 2024 Thorsten Brach. All rights reserved                                                                         
//                                                                           
//  Disclaimer:                                                                           
//    This project is provided without any guarantee and can be used for   
//    private and commercial purposes. Any commercial use is at the user’s 
//    own risk and responsibility.
//
// -------------------------------------------------------------------------
VAR_INPUT
  /// Set TRUE (default) to cyclically transmit data to the RC
  Enable            : BOOL;
END_VAR

VAR_OUTPUT
  /// Function is returning cyclic data from the RC
  Enabled           : BOOL;
  /// FB is being processed
  Busy              : BOOL;
  /// Cyclic input data of subprogram
  Data              : ARRAY[0..25] OF BYTE;
  
END_VAR

                  
                

METHOD PROTECTED OnCall
VAR_IN_OUT
  /// Robot assignment of function
  AxesGroup         : AxesGroup; 
END_VAR
                        
                      
END_METHOD
END_FUNCTION_BLOCK

/// Stops an active subprogram
FUNCTION_BLOCK StopSubprogramFB EXTENDS RobotLibraryBaseFB
// ------------------------------------------------------------------------- 
//  SRCI Robot Library                                                
// ------------------------------------------------------------------------- 
//                                                                           
//  Object:      StopSubprogramFB                                       
//  Author:      Thorsten Brach                                                
//  Date:        2024-06-01
//
//  Description:                                              
//   
//                                                                           
//  Copyright: 
//    (C) 2024 Thorsten Brach. All rights reserved                                                                         
//                                                                           
//  Disclaimer:                                                                           
//    This project is provided without any guarantee and can be used for   
//    private and commercial purposes. Any commercial use is at the user’s 
//    own risk and responsibility.
//
// -------------------------------------------------------------------------
VAR_INPUT
  /// Start of the command at the rising edge
  Execute           : BOOL;
  /// Processing mode
  ProcessingMode    : ProcessingMode;
  /// Defines how target subprogram is defined
  StopMode          : StopMode;
  /// JobID or InstanceID of target subprogram according to selected StopMode
  /// • Refers to StopMode 0 (Stop via JobID) and 1 (Stop via InstanceID).
  /// • -1: Invalid (default)
  TargetID          : UINT;
  /// Defines the target sequence in which the command will be executed
  SequenceFlag      : SequenceFlag;
  /// ID of associated trigger function:
  /// • 0: No Trigger (default) - No trigger related behavior
  /// • >0: Triggero - Start executing when the trigger function with the identical EmitterID is triggered.
  /// Always positive.
  /// For more information, see chapter 5.5.12 Triggers
  ListenerID        : SINT;
END_VAR

VAR_OUTPUT
  /// The command has been completed successfully
  Done               : BOOL;
  /// FB is being processed
  Busy               : BOOL;
  /// Command is transferred and confirmed by the RC
  CommandBuffered    : BOOL;
  /// The command was aborted by another command
  CommandAborted     : BOOL;
  /// TRUE, while command is interrupted during execution and can be continued.
  CommandInterrupted : BOOL;
  OriginID           : INT;
  /// Relates to ListenerID >0
  /// Number of successful trigger -based command invocations
  /// For more information refer to chapter 5.5.12.4.
  InvocationCounter  : USINT;
END_VAR

                  
                

METHOD PROTECTED OnCall
VAR_IN_OUT
  /// Robot assignment of function
  AxesGroup         : AxesGroup; 
END_VAR
                        
                      
END_METHOD
END_FUNCTION_BLOCK

/// Writes cyclic data of called subprogram
FUNCTION_BLOCK WriteCallSubprogramCyclicFB EXTENDS RobotLibraryBaseFB
// ------------------------------------------------------------------------- 
//  SRCI Robot Library                                                
// ------------------------------------------------------------------------- 
//                                                                           
//  Object:      WriteCallSubprogramCyclicFB                                       
//  Author:      Thorsten Brach                                                
//  Date:        2024-06-01
//
//  Description:                                              
//   
//                                                                           
//  Copyright: 
//    (C) 2024 Thorsten Brach. All rights reserved                                                                         
//                                                                           
//  Disclaimer:                                                                           
//    This project is provided without any guarantee and can be used for   
//    private and commercial purposes. Any commercial use is at the user’s 
//    own risk and responsibility.
//
// -------------------------------------------------------------------------
VAR_INPUT
  /// Set TRUE (default) to cyclically transmit data to the RC
  Enable            : BOOL;
  /// Cyclic input data of subprogram
  Data              : ARRAY[0..25] OF BYTE;
END_VAR

VAR_OUTPUT
  /// Data can now be written to the RC
  Enabled           : BOOL;
  /// FB is being processed
  Busy              : BOOL;
END_VAR

                  
                

METHOD PROTECTED OnCall
VAR_IN_OUT
  /// Robot assignment of function
  AxesGroup         : AxesGroup; 
END_VAR
                        
                      
END_METHOD
END_FUNCTION_BLOCK

/// "Action" that initiates specified events when triggered
FUNCTION_BLOCK ReactAtTriggerFB EXTENDS RobotLibraryBaseFB
// ------------------------------------------------------------------------- 
//  SRCI Robot Library                                                
// ------------------------------------------------------------------------- 
//                                                                           
//  Object:      ReactAtTriggerFB                                       
//  Author:      Thorsten Brach                                                
//  Date:        2024-06-01
//
//  Description:                                              
//   
//                                                                           
//  Copyright: 
//    (C) 2024 Thorsten Brach. All rights reserved                                                                         
//                                                                           
//  Disclaimer:                                                                           
//    This project is provided without any guarantee and can be used for   
//    private and commercial purposes. Any commercial use is at the user’s 
//    own risk and responsibility.
//
// -------------------------------------------------------------------------
VAR_INPUT
  /// Start of the command at the rising edge
  Execute                : BOOL;
  /// Processing mode
  ProcessingMode         : ProcessingMode;
  /// Defines RC’s and robot’s behavior when the"Action" is executed.
  ReactionMode           : TriggerReactionMode;
  /// ID of associated trigger function:
  /// • 0: Immediately (default) - Start executing this function immediately.
  /// • >0: Trigger -  Start executing, when the trigger function with the identical EmitterID is triggered.
  /// Always positive.
  /// For more information, see chapter 5.5.12 Triggers
  ListenerID             : SINT;
END_VAR
VAR_OUTPUT
  /// The command has been completed successfully
  Done                   : BOOL;
  /// FB is being processed
  Busy                   : BOOL;
  /// Command is transferred and confirmed by the RC
  CommandBuffered        : BOOL;
  /// Unique system-generated ID of the "Action" when the function is triggered.
  /// • >0: The "Action" is started by the trigger function with identical FollowID.
  /// • <0: The "Action" is stopped by the trigger function with identical FollowID.
  /// For more information see chapter 5.5.12.4 EmitterID, ListenerID, FollowID and OriginID
  OriginID               : INT;
  /// Relates to ListenerID >0
  /// Number of successful trigger -based command invocations
  /// For more information refer to chapter 5.5.12.4.
  InvocationCounter      : USINT;
END_VAR

                  
                

METHOD PROTECTED OnCall
VAR_IN_OUT
  /// Robot assignment of function
  AxesGroup         : AxesGroup; 
END_VAR
                        
                      
END_METHOD
END_FUNCTION_BLOCK

/// Trigger "Actions" based on incoming error event
FUNCTION_BLOCK SetTriggerErrorFB EXTENDS RobotLibraryBaseFB
// ------------------------------------------------------------------------- 
//  SRCI Robot Library                                                
// ------------------------------------------------------------------------- 
//                                                                           
//  Object:      SetTriggerErrorFB                                       
//  Author:      Thorsten Brach                                                
//  Date:        2024-06-01
//
//  Description:                                              
//   
//                                                                           
//  Copyright: 
//    (C) 2024 Thorsten Brach. All rights reserved                                                                         
//                                                                           
//  Disclaimer:                                                                           
//    This project is provided without any guarantee and can be used for   
//    private and commercial purposes. Any commercial use is at the user’s 
//    own risk and responsibility.
//
// -------------------------------------------------------------------------
VAR_INPUT
  /// Start of the command at the rising edge
  Execute                : BOOL;
  /// Processing mode
  ProcessingMode         : ProcessingMode;
  /// Defines error origin through which the associated Action will be triggered
  Mode                   : ErrorTriggerMode;
  /// Defines message codes through which the associated Action will be triggered (relates to Mode 6 and 7)
  MessageCodes           : ARRAY [0..15] OF DWORD;
  /// Defines if parametrization messages are included (relates to Mode 0 to 5)
  /// • FALSE (default): Do not include incorrect parametrization
  /// • TRUE: Include incorrect parametrization
  IncludeParameterValidation : BOOL;
  /// ID of associated trigger function:
  /// • 0: Immediately (default) - Start executing this function immediately.
  /// • >0: Trigger -  Start executing, when the trigger function with the identical EmitterID is triggered.
  /// Always positive.
  /// For more information, see chapter 5.5.12 Triggers
  ListenerID             : SINT;
  /// ID of the Action function that will be executed when the trigger condition is met
  /// • >0: Start Action        - Start executing the Action function with the identical ListenerID.
  /// • <0: Stop Action         - Stop executing the Action function with the identical ListenerID.
  /// •  0: Undefined (default) - If no EmitterID is defined, the function returns an error message
  /// For more information see chapter 5.5.12.4
  EmitterID              : SINT;  
END_VAR
VAR_OUTPUT
  /// The command has been completed successfully
  Done                   : BOOL;
  /// FB is being processed
  Busy                   : BOOL;
  /// Command is transferred and confirmed by the RC
  CommandBuffered        : BOOL;
  /// TRUE, when the monitoring of the input parameter values is active.
  MonitoringActive       : BOOL;
  /// Unique system-generated ID of the "Action" when the function is triggered.
  /// • >0: The "Action" is started by the trigger function with identical FollowID.
  /// • <0: The "Action" is stopped by the trigger function with identical FollowID.
  /// For more information see chapter 5.5.12.4 EmitterID, ListenerID, FollowID and OriginID
  OriginID               : INT;
  /// Relates to ListenerID >0
  /// Number of successful trigger -based command invocations
  /// For more information refer to chapter 5.5.12.4.
  InvocationCounter      : USINT;
  /// Unique system-generated ID of the trigger function when the function is called by user.
  /// For more information see chapter 5.5.12.4.
  FollowID               : DINT;
END_VAR

                  
                

METHOD PROTECTED OnCall
VAR_IN_OUT
  /// Robot assignment of function
  AxesGroup         : AxesGroup; 
END_VAR
                        
                      
END_METHOD
END_FUNCTION_BLOCK

/// Trigger "Actions" based on physical events (e.g. force limit reached)
FUNCTION_BLOCK SetTriggerLimitFB EXTENDS RobotLibraryBaseFB
// ------------------------------------------------------------------------- 
//  SRCI Robot Library                                                
// ------------------------------------------------------------------------- 
//                                                                           
//  Object:      SetTriggerLimitFB                                       
//  Author:      Thorsten Brach                                                
//  Date:        2024-06-01
//
//  Description:                                              
//   
//                                                                           
//  Copyright: 
//    (C) 2024 Thorsten Brach. All rights reserved                                                                         
//                                                                           
//  Disclaimer:                                                                           
//    This project is provided without any guarantee and can be used for   
//    private and commercial purposes. Any commercial use is at the user’s 
//    own risk and responsibility.
//
// -------------------------------------------------------------------------
VAR_INPUT
  /// Start of the command at the rising edge
  Execute                : BOOL;
  /// Processing mode
  ProcessingMode         : ProcessingMode;
  /// Specifies the trigger event by exceeding of the following limit values (one of the following options must be supported)
  TriggerMode            : TriggerModeLimit;
  /// Determines whether the start condition is evaluated or not.
  /// • FALSE: Start condition is not evaluated (default).
  /// • TRUE: Start condition is evaluated
  EvaluateStartCondition : BOOL;
  /// If the tolerance limits for the respective actual data values from the RC are exceeded, the Action function that will be executed.
  /// For "TriggerMode" 1, 2 and 4 the tolerance limits must be entered as follows:
  /// • [0..5]: relates to axes 1 to 6
  /// • [6..11]: relates to external axes 1 to 6.
  /// For "TriggerMode" 3 the tolerance limits must be entered as follows:
  /// • [0]: Following Error in mm.
  /// • [1..11]: Undefined and not relevant.
  /// For all array entries default: 999999
  Data_1                 : ARRAY[0..11] OF REAL;
  /// If the respective actual data values from the RC are under the defined limit, the Action function will be stopped.
  /// For "TriggerMode" 1, 2 and 4 the tolerance limits must be entered as follows:
  /// • [0..5]: relates to axes 1 to 6.
  /// • [6..11]: relates to external axes 1 to 6.
  /// For "TriggerMode" 3 the tolerance limits must be entered as follows:
  /// • [0]: Following Error in mm.
  /// • [1..11]: Undefined and not relevant.
  /// For all array entries default: 999999
  Data_2                 : ARRAY[0..11] OF REAL;
  /// ID of associated trigger function:
  /// • 0: Immediately (default) - Start executing this function immediately.
  /// • >0: Trigger -  Start executing, when the trigger function with the identical EmitterID is triggered.
  /// Always positive.
  /// For more information, see chapter 5.5.12 Triggers
  ListenerID             : SINT;
  /// ID of the Action function that will be executed when the trigger condition is met
  /// • >0: Start Action        - Start executing the Action function with the identical ListenerID.
  /// • <0: Stop Action         - Stop executing the Action function with the identical ListenerID.
  /// •  0: Undefined (default) - If no EmitterID is defined, the function returns an error message
  /// For more information see chapter 5.5.12.4
  EmitterID              : SINT;  
END_VAR
VAR_OUTPUT
  /// The command has been completed successfully
  Done                   : BOOL;
  /// TRUE, while the following outputs return valid values:
  /// • Data
  Valid                  : BOOL;
  /// FB is being processed
  Busy                   : BOOL;
  /// Command is transferred and confirmed by the RC
  CommandBuffered        : BOOL;
  /// The respective actual data values from the RC that depend on "TriggerMode".
  Data                   : ARRAY [0..11] OF REAL;  
  /// TRUE, when the monitoring of the input parameter values is active.
  MonitoringActive       : BOOL;
  /// Unique system-generated ID of the "Action" when the function is triggered.
  /// • >0: The "Action" is started by the trigger function with identical FollowID.
  /// • <0: The "Action" is stopped by the trigger function with identical FollowID.
  /// For more information see chapter 5.5.12.4 EmitterID, ListenerID, FollowID and OriginID
  OriginID               : INT;
  /// Relates to ListenerID >0
  /// Number of successful trigger -based command invocations
  /// For more information refer to chapter 5.5.12.4.
  InvocationCounter      : USINT;
  /// Unique system-generated ID of the trigger function when the function is called by user.
  /// For more information see chapter 5.5.12.4.
  FollowID               : DINT;
END_VAR

                  
                

METHOD PROTECTED OnCall
VAR_IN_OUT
  /// Robot assignment of function
  AxesGroup         : AxesGroup; 
END_VAR
                        
                      
END_METHOD
END_FUNCTION_BLOCK

/// Trigger an action based on a motion related parameter (e.g. progress of trajectory)
FUNCTION_BLOCK SetTriggerMotionFB EXTENDS RobotLibraryBaseFB
// ------------------------------------------------------------------------- 
//  SRCI Robot Library                                                
// ------------------------------------------------------------------------- 
//                                                                           
//  Object:      SetTriggerMotionFB                                       
//  Author:      Thorsten Brach                                                
//  Date:        2024-06-01
//
//  Description:                                              
//   
//                                                                           
//  Copyright: 
//    (C) 2024 Thorsten Brach. All rights reserved                                                                         
//                                                                           
//  Disclaimer:                                                                           
//    This project is provided without any guarantee and can be used for   
//    private and commercial purposes. Any commercial use is at the user’s 
//    own risk and responsibility.
//
// -------------------------------------------------------------------------
VAR_INPUT
  /// Start of the command at the rising edge
  Execute                : BOOL;
  /// Processing mode
  ProcessingMode         : ProcessingMode;
  ///Defines the trigger condition on which the related Action function will be started:
  TriggerMode_1          : TriggerCondition;
  /// This parameter depends on the input parameter "TriggerMode_1":
  /// • 1: Distance value of trajectory in %.
  /// • 2: Distance value of trajectory in mm.
  /// • 3: TCP velocity value of reference velocity in %
  /// • 4: TCP velocity value of reference velocity in mm.
  /// • 5: Time in ms
  /// The value of the parameter must be positive  
  TriggerParameter_1     : REAL;
  ///Defines the trigger condition on which the related Action function will be started:
  TriggerMode_2          : TriggerCondition;
  /// This parameter depends on the input parameter "TriggerMode_1":
  /// • 1: Distance value of trajectory in %. 
  /// • 2: Distance value of trajectory in mm.
  /// • 3: TCP velocity value of reference velocity in %
  /// • 4: TCP velocity value of reference velocity in mm.
  /// • 5: Time in ms
  /// The value of the parameter must be positive  
  TriggerParameter_2     : REAL;
  /// ID of associated trigger function:
  /// • 0: Immediately (default) - Start executing this function immediately.
  /// • >0: Trigger -  Start executing, when the trigger function with the identical EmitterID is triggered.
  /// Always positive.
  /// For more information, see chapter 5.5.12 Triggers
  ListenerID             : SINT;
  /// ID of the Action function that will be executed when the trigger condition is met
  /// • >0: Start Action        - Start executing the Action function with the identical ListenerID.
  /// • <0: Stop Action         - Stop executing the Action function with the identical ListenerID.
  /// •  0: Undefined (default) - If no EmitterID is defined, the function returns an error message
  /// For more information see chapter 5.5.12.4
  EmitterID              : SINT;  
END_VAR

VAR_OUTPUT
  /// The command has been completed successfully
  Done                   : BOOL;
  /// FB is being processed
  Busy                   : BOOL;
  /// Command is transferred and confirmed by the RC
  CommandBuffered        : BOOL;
  /// TRUE, when the monitoring of the input parameter values is active.
  MonitoringActive       : BOOL;
  /// Unique system-generated ID of the "Action" when the function is triggered.
  /// • >0: The "Action" is started by the trigger function with identical FollowID.
  /// • <0: The "Action" is stopped by the trigger function with identical FollowID.
  /// For more information see chapter 5.5.12.4 EmitterID, ListenerID, FollowID and OriginID
  OriginID               : INT;
  /// Relates to ListenerID >0
  /// Number of successful trigger -based command invocations
  /// For more information refer to chapter 5.5.12.4.
  InvocationCounter      : USINT;
  /// Unique system-generated ID of the trigger function when the function is called by user.
  /// For more information see chapter 5.5.12.4.
  FollowID               : DINT;
END_VAR

                  
                

METHOD PROTECTED OnCall
VAR_IN_OUT
  /// Robot assignment of function
  AxesGroup         : AxesGroup; 
END_VAR
                        
                      
END_METHOD
END_FUNCTION_BLOCK

/// Trigger "Actions" based on I/O related events (e.g. change of DI’s state)
FUNCTION_BLOCK SetTriggerRegisterFB EXTENDS RobotLibraryBaseFB
// ------------------------------------------------------------------------- 
//  SRCI Robot Library                                                
// ------------------------------------------------------------------------- 
//                                                                           
//  Object:      SetTriggerRegisterFB                                       
//  Author:      Thorsten Brach                                                
//  Date:        2024-06-01
//
//  Description:                                              
//   
//                                                                           
//  Copyright: 
//    (C) 2024 Thorsten Brach. All rights reserved                                                                         
//                                                                           
//  Disclaimer:                                                                           
//    This project is provided without any guarantee and can be used for   
//    private and commercial purposes. Any commercial use is at the user’s 
//    own risk and responsibility.
//
// -------------------------------------------------------------------------
VAR_INPUT
  /// Start of the command at the rising edge
  Execute                : BOOL;
  /// Processing mode
  ProcessingMode         : ProcessingMode;
  /// Specifies the trigger event according to Table 6-574.
  /// For more information about registers on the RC see chapters 6.4.4 and 6.4.5.
  TriggerMode            : TriggerModeIo;
  /// Determines whether the start condition is evaluated or not.
  /// • FALSE: Start condition is not evaluated (default).
  /// • TRUE: Start condition is evaluated. 
  EvaluateStartCondition : BOOL;
  /// Depending on "TriggerMode":
  /// • Digital (refers to "TriggerMode" 10-13, 20-23): Specifies the desired byte address of the input or output signal that shall be read.
  /// • Analog/Integer/Real (refers to "TriggerMode" 30-37, 40-47, 50-57, 60- 67): Specifies the target values that shall be read.
  /// For more information about registers refer to Figure 6-206.
  Index                  : USINT;
  /// Depending on "TriggerMode":
  /// • Digital (refers to TriggerMode 10-13,20-23): Specifies the desired bit address of the input or output signal that shall be read.
  /// • Analog/Integer/Real (refers to TriggerMode 30-37, 40-47, 50-57, 60- 67): Not relevant and deactivated for user input.
  /// For more information about registers refer to Figure 6-206
  BitIndex               : USINT;
  /// Reference integer value, for triggering the Action function with the EmitterID.
  /// • Relates to "TriggerMode" 50-57
  IntValue               : ARRAY[1..2] OF INT;
  /// Reference real value, analog input or output value, for triggering the Action function with the EmitterID.
  /// • Relates to "TriggerMode" 30-37, 40-47,60-67
  RealValue              : ARRAY[1..2] OF REAL;
  /// ID of associated trigger function:
  /// • 0: Immediately (default). - Start executing this function immediately.
  /// • >0: Trigger - Start executing, when the trigger function with the identical EmitterID is triggered.
  /// Always positive.
  /// For more information, see chapter 5.5.12 Triggers
  ListenerID             : SINT;
  /// ID of the Action function that will be executed when the trigger condition is met
  /// • >0: Start Action        - Start executing the Action function with the identical ListenerID.
  /// • <0: Stop Action         - Stop executing the Action function with the identical ListenerID.
  /// •  0: Undefined (default) - If no EmitterID is defined, the function returns an error message
  /// For more information see chapter 5.5.12.4
  EmitterID              : SINT;
END_VAR
VAR_OUTPUT
  /// The command has been completed successfully
  Done                   : BOOL;
  /// FB is being processed
  Busy                   : BOOL;
  /// Command is transferred and confirmed by the RC
  CommandBuffered        : BOOL;
  /// TRUE, when the monitoring of the input parameter values is active.
  MonitoringActive       : BOOL;
  /// Unique system-generated ID of the "Action" when the function is triggered.
  /// • >0: The "Action" is started by the trigger function with identical FollowID.
  /// • <0: The "Action" is stopped by the trigger function with identical FollowID.
  /// For more information see chapter 5.5.12.4 EmitterID, ListenerID, FollowID and OriginID
  OriginID               : INT;
  /// Relates to ListenerID >0
  /// Number of successful trigger -based command invocations
  /// For more information refer to chapter 5.5.12.4.
  InvocationCounter      : USINT;
  /// Unique system-generated ID of the trigger function when the function is called by user.
  /// For more information see chapter 5.5.12.4.
  FollowID               : DINT;
END_VAR

                  
                

METHOD PROTECTED OnCall
VAR_IN_OUT
  /// Robot assignment of function
  AxesGroup         : AxesGroup; 
END_VAR
                        
                      
END_METHOD
END_FUNCTION_BLOCK

/// Trigger "Actions" based on physical events (e.g. force limit reached)
FUNCTION_BLOCK SetTriggerUserFB EXTENDS RobotLibraryBaseFB
// ------------------------------------------------------------------------- 
//  SRCI Robot Library                                                
// ------------------------------------------------------------------------- 
//                                                                           
//  Object:      SetTriggerUserFB                                       
//  Author:      Thorsten Brach                                                
//  Date:        2024-06-01
//
//  Description:                                              
//   
//                                                                           
//  Copyright: 
//    (C) 2024 Thorsten Brach. All rights reserved                                                                         
//                                                                           
//  Disclaimer:                                                                           
//    This project is provided without any guarantee and can be used for   
//    private and commercial purposes. Any commercial use is at the user’s 
//    own risk and responsibility.
//
// -------------------------------------------------------------------------
VAR_INPUT
  /// Start of the command at the rising edge
  Execute                : BOOL;
  /// Processing mode
  ProcessingMode         : ProcessingMode;
  /// Defines the target sequence in which the command will be executed
  SequenceFlag           : SequenceFlag;
  /// ID of the Action function that will be executed when the trigger condition is met
  /// • >0: Start Action        - Start executing the Action function with the identical ListenerID.
  /// • <0: Stop Action         - Stop executing the Action function with the identical ListenerID.
  /// •  0: Undefined (default) - If no EmitterID is defined, the function returns an error message
  /// For more information see chapter 5.5.12.4
  EmitterID              : SINT;  
END_VAR
VAR_OUTPUT
  /// The command has been completed successfully
  Done                   : BOOL;
  /// FB is being processed
  Busy                   : BOOL;
  /// Command is transferred and confirmed by the RC
  CommandBuffered        : BOOL;
  /// The command was aborted by another command
  CommandAborted         : BOOL;
  /// TRUE, while command is interrupted during execution and can be continued.
  CommandInterrupted     : BOOL;
  /// Unique system-generated ID of the trigger function when the function is called by user.
  /// For more information see chapter 5.5.12.4.
  FollowID               : DINT;
END_VAR

                  
                

METHOD PROTECTED OnCall
VAR_IN_OUT
  /// Robot assignment of function
  AxesGroup         : AxesGroup; 
END_VAR
                        
                      
END_METHOD
END_FUNCTION_BLOCK

/// Wait to process next command in sequence until trigger signal is received
FUNCTION_BLOCK WaitForTriggerFB EXTENDS RobotLibraryBaseFB
// ------------------------------------------------------------------------- 
//  SRCI Robot Library                                                
// ------------------------------------------------------------------------- 
//                                                                           
//  Object:      WaitForTriggerFB                                       
//  Author:      Thorsten Brach                                                
//  Date:        2024-06-01
//
//  Description:                                              
//   
//                                                                           
//  Copyright: 
//    (C) 2024 Thorsten Brach. All rights reserved                                                                         
//                                                                           
//  Disclaimer:                                                                           
//    This project is provided without any guarantee and can be used for   
//    private and commercial purposes. Any commercial use is at the user’s 
//    own risk and responsibility.
//
// -------------------------------------------------------------------------
VAR_INPUT
  /// Start of the command at the rising edge
  Execute                : BOOL;
  /// Processing mode
  ProcessingMode         : ProcessingMode;
  ///  Defines the time at which the trigger can be reacted to
  /// • 0: Conditional - Trigger signal accepted as soon as the function is BUFFERED
  /// • 1: Absolute - Trigger signal accepted as soon as the function is ACTIVE
  ConditionalWait        : BOOL;
  /// Defines the target sequence in which the command will be executed
  SequenceFlag           : SequenceFlag;
  /// ID of associated trigger function:
  /// • 0: Immediately (default) - Start executing this function immediately.
  /// • >0: Trigger -  Start executing, when the trigger function with the identical EmitterID is triggered.
  /// Always positive.
  /// For more information, see chapter 5.5.12 Triggers
  ListenerID             : SINT;
END_VAR
VAR_OUTPUT
  /// The command has been completed successfully
  Done                   : BOOL;
  /// FB is being processed
  Busy                   : BOOL;
  /// Command is transferred and confirmed by the RC
  CommandBuffered        : BOOL;
  /// Command is currently processed by the active sequence, takes control of the motion of the according axis group and is waiting for Trigger.
  Active                 : BOOL;
  /// The command was aborted by another command
  CommandAborted         : BOOL;
  /// TRUE, while command is interrupted during execution and can be continued.
  CommandInterrupted     : BOOL;
  /// Unique system-generated ID of the "Action" when the function is triggered.
  /// • >0: The "Action" is started by the trigger function with identical FollowID.
  /// • <0: The "Action" is stopped by the trigger function with identical FollowID.
  /// For more information see chapter 5.5.12.4 EmitterID, ListenerID, FollowID and OriginID
  OriginID               : INT;
  /// Relates to ListenerID >0
  /// Number of successful trigger -based command invocations
  /// For more information refer to chapter 5.5.12.4.
  InvocationCounter      : USINT;
END_VAR

                  
                

METHOD PROTECTED OnCall
VAR_IN_OUT
  /// Robot assignment of function
  AxesGroup         : AxesGroup; 
END_VAR
                        
                      
END_METHOD
END_FUNCTION_BLOCK

/// Write analog output of RC
FUNCTION_BLOCK WriteAnalogOutputFB EXTENDS RobotLibraryBaseFB
// ------------------------------------------------------------------------- 
//  SRCI Robot Library                                                
// ------------------------------------------------------------------------- 
//                                                                           
//  Object:      WriteAnalogOutputFB                                       
//  Author:      Thorsten Brach                                                
//  Date:        2024-06-01
//
//  Description:                                              
//   
//                                                                           
//  Copyright: 
//    (C) 2024 Thorsten Brach. All rights reserved                                                                         
//                                                                           
//  Disclaimer:                                                                           
//    This project is provided without any guarantee and can be used for   
//    private and commercial purposes. Any commercial use is at the user’s 
//    own risk and responsibility.
//
// -------------------------------------------------------------------------
VAR_INPUT
  /// Start of the command at the rising edge
  Execute            : BOOL;
  /// Processing Mode
  ProcessingMode     : ProcessingMode;
  /// Number of the analog input 1..32
  Index              : USINT;
  /// Value of analog output
  Value              : REAL;
  /// Unit of set Value:
  Unit               : UnitType;
  /// Set TRUE to prioritize the execution of this command in the defined target sequence.             
  HighPriority       : BOOL;
  /// Defines the target sequence in which the command will be executed
  SequenceFlag       : SequenceFlag;
  /// ID of associated trigger function:
  /// •  0: No Trigger (default)  No trigger related behavior
  /// • >0: Trigger - Start executing when the trigger function with the identical EmitterID is triggered.
  /// Always positive.
  /// For more information, see chapter 5.5.12 Triggers
  ListenerID         : SINT;
END_VAR
VAR_OUTPUT
  /// The command has been completed successfully
  Done               : BOOL;
  /// FB is being processed
  Busy               : BOOL;
  /// Command is transferred and confirmed by the RC
  CommandBuffered    : BOOL;
  /// The command was aborted by another command.
  CommandAborted     : BOOL;
  /// TRUE, while command is interrupted during execution and can be continued
  CommandInterrupted : BOOL;
  /// Receiving of input parameter values has been acknowledged by RC
  ParameterAccepted  : BOOL;
  /// Unique system-generated ID of the "Action" when the function is triggered.
  /// • >0: The "Action" is started by the trigger function with identical FollowID.
  /// • <0: The "Action" is stopped by the trigger function with identical FollowID.
  /// For more information see chapter 5.5.12.4.
  OriginID           : USINT;
  /// Relates to ListenerID >0 
  /// Number of successful trigger -based command invocations
  /// For more information refer to chapter 5.5.12.4.
  InvocationCounter  : USINT;
END_VAR

                  
                

METHOD PROTECTED OnCall
VAR_IN_OUT
  /// Robot assignment of function
  AxesGroup         : AxesGroup; 
END_VAR
                        
                      
END_METHOD
END_FUNCTION_BLOCK

/// Write digital output group of RC
FUNCTION_BLOCK WriteDigitalOutputsFB EXTENDS RobotLibraryBaseFB
// ------------------------------------------------------------------------- 
//  SRCI Robot Library                                                
// ------------------------------------------------------------------------- 
//                                                                           
//  Object:      WriteDigitalOutputsFB                                       
//  Author:      Thorsten Brach                                                
//  Date:        2024-06-01
//
//  Description:                                              
//   
//                                                                           
//  Copyright: 
//    (C) 2024 Thorsten Brach. All rights reserved                                                                         
//                                                                           
//  Disclaimer:                                                                           
//    This project is provided without any guarantee and can be used for   
//    private and commercial purposes. Any commercial use is at the user’s 
//    own risk and responsibility.
//
// -------------------------------------------------------------------------
VAR_INPUT
  /// Start of the command at the rising edge
  Execute            : BOOL;
  /// Processing Mode
  ProcessingMode     : ProcessingMode;
  /// Specifies the desired byte addresses that shall be read
  Index              : ARRAY[0..4] OF USINT;
  /// Specifies which outputs may be written
  OutputBitmask      : ARRAY[0..4] OF BYTE;
  /// Array value of Digital Output
  Values             : ARRAY[0..4] OF BYTE;
  /// Set TRUE to prioritize the execution of this command in the defined target sequence.             
  HighPriority       : BOOL;
  /// Defines the target sequence in which the command will be executed
  SequenceFlag       : SequenceFlag;
  /// ID of associated trigger function:
  /// •  0: No Trigger (default)  No trigger related behavior
  /// • >0: Trigger - Start executing when the trigger function with the identical EmitterID is triggered.
  /// Always positive.
  /// For more information, see chapter 5.5.12 Triggers
  ListenerID         : SINT;
END_VAR
VAR_OUTPUT
  /// The command has been completed successfully
  Done               : BOOL;
  /// FB is being processed
  Busy               : BOOL;
  /// Command is transferred and confirmed by the RC
  CommandBuffered    : BOOL;
  /// The command was aborted by another command.
  CommandAborted     : BOOL;
  /// TRUE, while command is interrupted during execution and can be continued
  CommandInterrupted : BOOL;
  /// Receiving of input parameter values has been acknowledged by RC
  ParameterAccepted  : BOOL;
  /// Unique system-generated ID of the "Action" when the function is triggered.
  /// • >0: The "Action" is started by the trigger function with identical FollowID.
  /// • <0: The "Action" is stopped by the trigger function with identical FollowID.
  /// For more information see chapter 5.5.12.4.
  OriginID           : USINT;
  /// Relates to ListenerID >0 
  /// Number of successful trigger -based command invocations
  /// For more information refer to chapter 5.5.12.4.
  InvocationCounter  : USINT;
END_VAR

                  
                

METHOD PROTECTED OnCall
VAR_IN_OUT
  /// Robot assignment of function
  AxesGroup         : AxesGroup; 
END_VAR
                        
                      
END_METHOD
END_FUNCTION_BLOCK

